(* Logix 5000 project; controller Carpenter_Meter_SCP vendor 1 type 14 code 217 rev 31.11; software revision 31.01; part 6 of 7 *)
(* tags used below, declared in another part *)
   AlwaysOff : BOOL;   // Always Off Bit
   CAR100_Flowpath : BOOL;   // Carpenter MLV CAR100 Flow Path (1=OK)
   CAR100_High_Pressure_SD : BOOL;   // Carpenter MLV CAR100 High Pressure Shutdown Status
   Carpenter_ISD_Command : BOOL;   // Carpenter/Hereford ISD Command from OCC (Through Pawnee)
   Carpenter_to_Pawnee_OK : BOOL;   // Carpenter to Pawnee Flow Path Permissive
   CC_Cust1_Flow_Permissive : BOOL;   // Customer #1 (MS8800) Flow Permissive to OCC
   CC_Cust1_Hi_WIOM : BOOL;   // Customer #1 High Water % Alarm to OCC
   CC_Cust1_Pump_Running : BOOL;   // Customer #1 (MS8800) Pump Running Status to OCC
   CC_Cust1_Ready : BOOL;   // Customer #1 (MS8800) Ready Status to OCC
   CC_Cust1_Shutin_Timer : REAL;   // Customer #1 Shutin Reset Time Left to OCC
   CC_Cust1_WIOM_Shutin : BOOL;   // Customer #1 Shutin Due to High High Water in Oil Monitor Alarm to OCC
   CC_Cust5_Flow_Permissive : BOOL;   // Customer #5 (MS8840) Flow Permissive to OCC
   CC_Cust5_Ready : BOOL;   // Customer #5 (MS8840) Ready Status to OCC
   CC_MS8800_Biocide_Flow : REAL;   // Meter Skid MS-8800 Biocide Flow Rate
   CC_MS8800_Biocide_Flow_SP : REAL;   // Meter Skid MS-8800 Biocide Flow Rate Setpoint
   CC_MS8800_CustPress : OCC_Analog;   // Meter Skid MS-8800 Customer Inlet Pressure to OCC
   CC_MS8810_CustPress : OCC_Analog;   // Meter Skid MS-8810 Customer Inlet Pressure to OCC
   CC_MS8820_CustPress : OCC_Analog;   // Meter Skid MS-8820 Customer Inlet Pressure to OCC
   CC_MS8830_CustPress : OCC_Analog;   // Meter Skid MS-8830 Customer Inlet Pressure to OCC
   CC_MS8840_Biocide_Flow : REAL;   // Meter Skid MS-8800 Biocide Flow Rate
   CC_MS8840_Biocide_Flow_SP : REAL;   // Meter Skid MS-8800 Biocide Flow Rate Setpoint
   CC_MS8840_CustPress : OCC_Analog;   // Meter Skid MS-8840 Customer Inlet Pressure to OCC
   CC_Pawnee_Flow_Path : BOOL;   // Flow Path to Pawnee
   CC_PV_0001 : OCC_CV;   // PV-0001
   CC_PV_0001_Flow_SP : DINT;   // Meter Skid MS8800 Inlet Control Valve Flow Setpoint
   CC_PV_0001_Press_SP : DINT;   // Meter Skid MS8800 Inlet Control Valve Press Setpoint
   CC_PV_0041 : OCC_CV;   // PV-0041
   CC_PV_0041_Flow_SP : DINT;   // Meter Skid MS8840 Inlet Control Valve Flow Setpoint
   CC_PV_0041_Press_SP : DINT;   // Meter Skid MS8800 Inlet Control Valve Press Setpoint
   CC_STA_Stop : BOOL;   // Station Stop Request Command from OCC
   CC_XI_0021 : BOOL;   // FGP Main PLC 24VDC Failure to OCC
   CC_XI_8800B : BOOL;   // MS8800 FGP 24VDC Failure to OCC
   CC_XI_8840B : BOOL;   // MS8840 FGP 24VDC Failure to OCC
   CC_YI_6000 : BOOL;   // UPS-6000 Utility Power Loss to OCC
   CC_YI_6001 : BOOL;   // UPS-6000 Fault
   cmd_reset_tmr : TIMER[8];   // General Use HMI Command Reset Timer
   Cust1_WIOM_Alarm : BOOL;   // Customer 1 WIOM Alarm
   Cust1_WIOM_Reset_Tmr : TIMER;   // Customer 1 Reset Timer for a WIOM Shutin
   Customer1_Flowpath_OK : BOOL;   // Customer #1 Flowpath Permissive (1 = OK)
   Customer1_Pump_Status : BOOL;   // Customer #1 Pump Running Status
   Customer1_Ready_Status : BOOL;   // Customer #1 Ready Status
   Customer5_Flowpath_OK : BOOL;   // Customer #5 Flowpath Permissive (1 = OK)
   Customer5_Ready_Status : BOOL;   // Customer #4 Ready Status
   fgp_deactivate_keysw : BOOL;   // Fire and Gas System Deactivated through Key Switch
   FGP_ESD : TGE_Alarm;   // ESD Shutdown from FGP (HS-0020A)
   FGP_Fire_Det : TGE_Alarm;   // Fire Shutdown from FGP (YSHH-0022)
   FGP_Gas_Det : TGE_Alarm;   // Hi Gas Shutdown from FGP (ASHH-0021)
   fgp_panel_reset : BOOL;   // FGP Panel Reset Pushbutton
   Hereford_Flowpath : BOOL;   // Pawnee Terminal Flow Path (1=OK)
   Hereford_High_Pressure_SD : BOOL;   // Hereford High Pressure Shutdown Status
   Hereford_OCC_HB_FAIL : BOOL;   // Pawnee High Pressure Shutdown Status
   HRF100_Flowpath : BOOL;   // Hereford MLV HRF100 Flow Path (1=OK)
   HRF100_High_Pressure_SD : BOOL;   // Hereford MLV HRF100 High Pressure Shutdown Status
   Main_FGP_24VDC_Fail : TGE_Alarm;   // Main PLC FGP 24VDC Fail (XS-0021)
   MS8800_Biocide_Flow_Fdbk_AOI : TGE_AI;   // Meter Skid MS-8800 Biocide Injection Rate Feedback
   MS8800_Biocide_Flow_SP : REAL;   // Meter Skid MS-8800 Biocide Flow Rate Gal/Day
   MS8800_Cust_Press : TGE_AI_UDT;   // Meter Skid MS-8800 Customer Inlet Pressure (Communicated from Cust)
   MS8800_FGP_24VDC_Fail : TGE_Alarm;   // Meter Skid MS-8800 FGP 24VDC Fail (XS-8800B)
   MS8800_Flow_Control : PID;   // Meter Skid MS8800 Flow Rate P&ID
   MS8800_Inlet_Press_Control : PID;   // Meter Skid MS8800 Customer Inlet Pressure P&ID
   MS8800_PCV_Pos_AOI : TGE_AI;   // Meter Skid MS-8800 Pressure Control Valve - Position Feedback (PCV-0001)
   MS8800_WIOM_Alarm : AnalogAlm;   // MS8800 Water In Oil Monitor Alarm (Setpoint Dictated by Tarrif)
   MS8840_Biocide_Flow_Fdbk_AOI : TGE_AI;   // Meter Skid MS-8840 Biocide Injection Rate Feedback
   MS8840_Biocide_Flow_SP : REAL;   // Meter Skid MS-8840 Biocide Flow Rate Gal/Day
   MS8840_Cust_Press : TGE_AI_UDT;   // Meter Skid MS-8840 Customer Inlet Pressure (Communicated from Cust)
   MS8840_FGP_24VDC_Fail : TGE_Alarm;   // Meter Skid MS-8840 FGP 24VDC Fail (XS-8840B)
   MS8840_Flow_Control : PID;   // Meter Skid MS8840 Flow Rate P&ID
   MS8840_Inlet_Press_Control : PID;   // Meter Skid MS8840 Customer Inlet Pressure P&ID
   MS8840_PCV_Pos_AOI : TGE_AI;   // Meter Skid MS-8840 Pressure Control Valve - Position Feedback (PCV-0041)
   ons_gen_use : BOOL[64];
   ovrd_disch_press : Override;   // Discharge Pressure Override
   ovrd_esd : Override;   // ESD Override
   ovrd_fire : Override;   // Fire Override
   ovrd_gas : Override;   // Gas Override
   Pawnee_ESD : BOOL;   // Pawnee Terminal ESD Signal (1=OK, 0 = ESD Active)
   Pawnee_Flowpath : BOOL;   // Pawnee Terminal Flow Path (1=OK)
   Pawnee_High_Pressure_SD : BOOL;   // Pawnee High Pressure Shutdown Status
   Pawnee_OCC_HB_FAIL : BOOL;   // Pawnee OCC HB Fail
   PV0001_Malf : TGE_Alarm;   // PV0001 Malfunction Alarm
   PV0001_Pos_Cmd : REAL;   // PCV-0001 Position Command
   PV0041_Malf : TGE_Alarm;   // PV0041 Malfunction Alarm
   PV0041_Pos_Cmd : REAL;   // PCV-0041 Position Command
   SCADA_HB_Fail_Alm : TGE_Alarm;   // SCADA Hearbeat Failure Alarm
   Sta_Stat : StaStatus;
   sta_stop : StaStartStop;   // Station Stop
   sta_stop_vlv_req : BOOL;   // Station Stop Valve Close Request
   Station_Disch_Press : TGE_AI_UDT;   // Station Discharge Pressure - Launcher Skid (PIT-1101)
   Test : BOOL;
   TU3000_HiHi_Lvl : TGE_Alarm;   // Sump Tank (TU-3000) Hi Hi Level Switch (LSHH-3000)
   TU3100_HiHi_Lvl : TGE_Alarm;   // Sump Tank (TU-3100) Hi Hi Level Switch (LSHH-3100)
   UPS_Fault : TGE_Alarm;   // UPS-6000 Fault (YS-6001)
   UPS_Online : TGE_Alarm;   // UPS-6000 Loss of AC Feed (YS-6000)
   valve_failure : BOOL;   // Valve Failure Override
   XV_0001 : BaseVLVLiquid;   // XV-0001
   XV_0041 : BaseVLVLiquid;   // XV-0041
   XV_1100 : BaseVLVLiquid;   // XV-1100
   XV_1101 : BaseVLVLiquid;   // XV-1101
(* OCC_Comms, continued *)

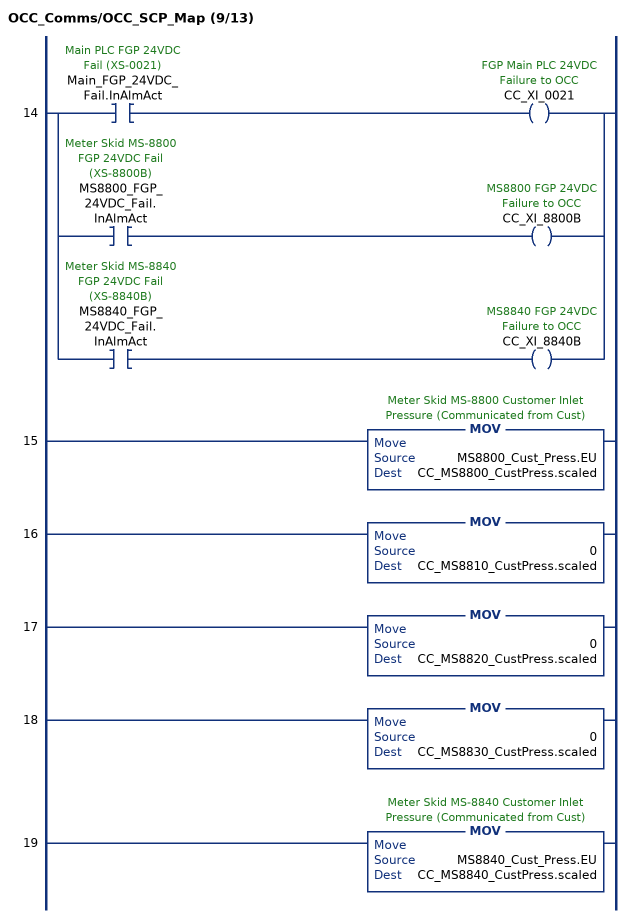
   [picture p98: OCC_Comms/OCC_SCP_Map rungs 14-19]
   14: [XIC(Main_FGP_24VDC_Fail.InAlmAct) OTE(CC_XI_0021) ,XIC(MS8800_FGP_24VDC_Fail.InAlmAct) OTE(CC_XI_8800B) ,XIC(MS8840_FGP_24VDC_Fail.InAlmAct) OTE(CC_XI_8840B) ];
   15: MOV(MS8800_Cust_Press.EU,CC_MS8800_CustPress.scaled);
   16: MOV(0,CC_MS8810_CustPress.scaled);
   17: MOV(0,CC_MS8820_CustPress.scaled);
   18: MOV(0,CC_MS8830_CustPress.scaled);
   19: MOV(MS8840_Cust_Press.EU,CC_MS8840_CustPress.scaled);
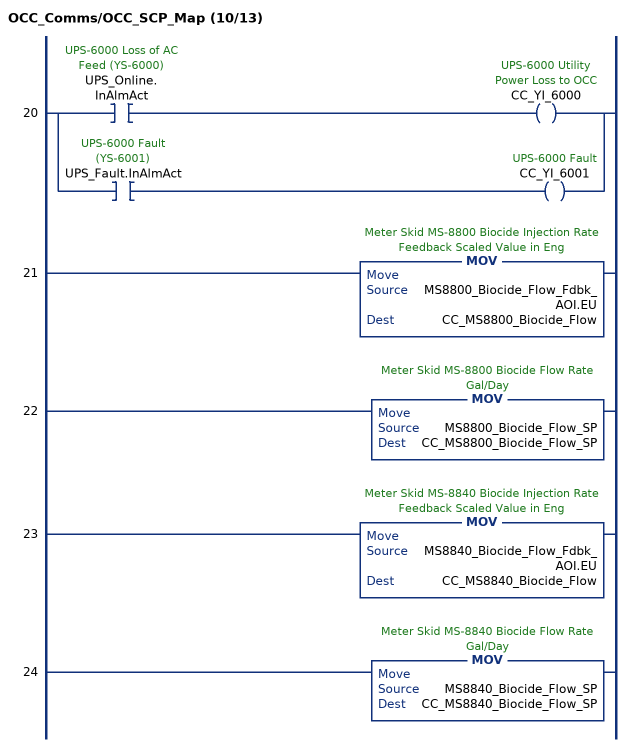
   20: [XIC(UPS_Online.InAlmAct) OTE(CC_YI_6000) ,XIC(UPS_Fault.InAlmAct) OTE(CC_YI_6001) ];
   21: MOV(MS8800_Biocide_Flow_Fdbk_AOI.EU,CC_MS8800_Biocide_Flow);
   22: MOV(MS8800_Biocide_Flow_SP,CC_MS8800_Biocide_Flow_SP);
   23: MOV(MS8840_Biocide_Flow_Fdbk_AOI.EU,CC_MS8840_Biocide_Flow);
   24: MOV(MS8840_Biocide_Flow_SP,CC_MS8840_Biocide_Flow_SP);
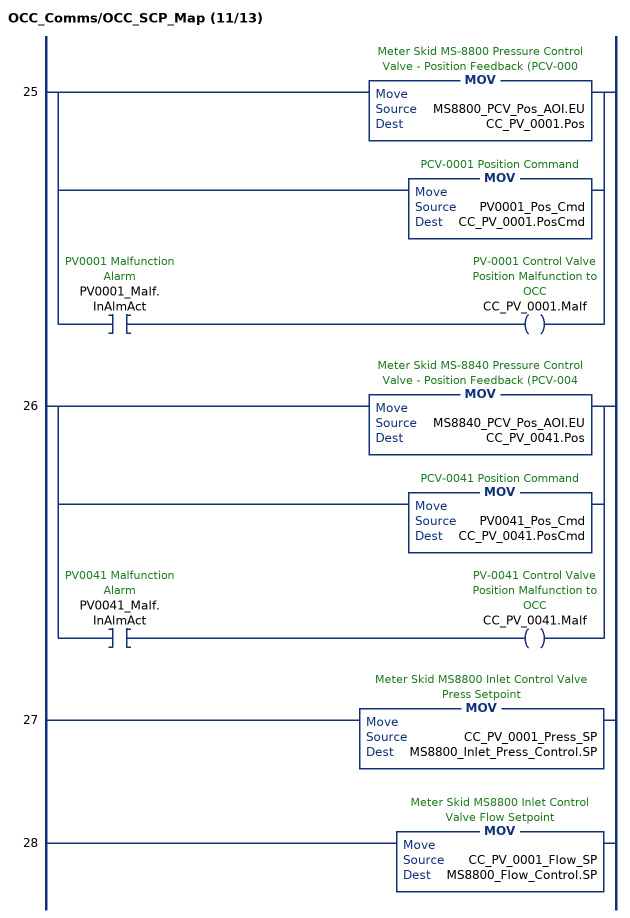
   25: [MOV(MS8800_PCV_Pos_AOI.EU,CC_PV_0001.Pos) ,MOV(PV0001_Pos_Cmd,CC_PV_0001.PosCmd) ,XIC(PV0001_Malf.InAlmAct) OTE(CC_PV_0001.Malf) ];
   26: [MOV(MS8840_PCV_Pos_AOI.EU,CC_PV_0041.Pos) ,MOV(PV0041_Pos_Cmd,CC_PV_0041.PosCmd) ,XIC(PV0041_Malf.InAlmAct) OTE(CC_PV_0041.Malf) ];
   27: MOV(CC_PV_0001_Press_SP,MS8800_Inlet_Press_Control.SP);
   28: MOV(CC_PV_0001_Flow_SP,MS8800_Flow_Control.SP);
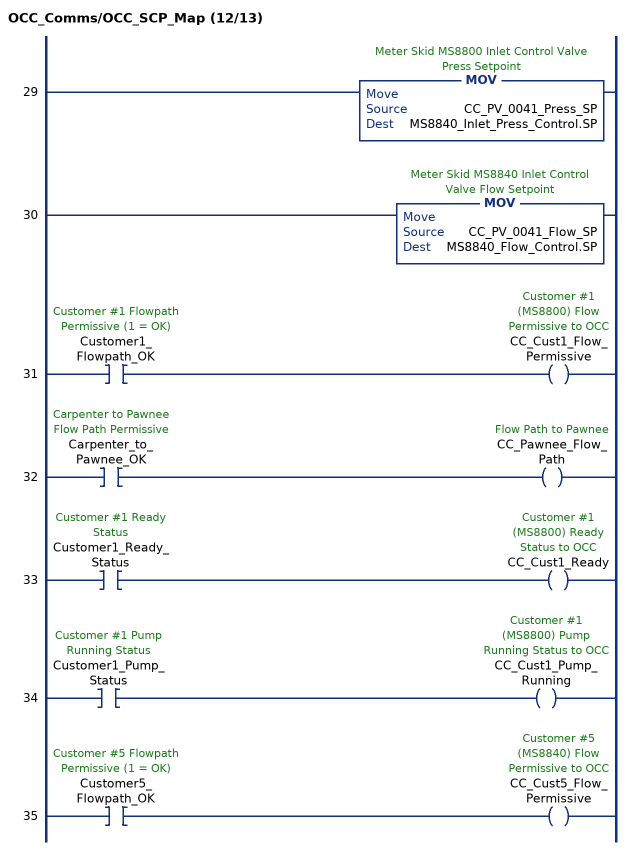
   29: MOV(CC_PV_0041_Press_SP,MS8840_Inlet_Press_Control.SP);
   30: MOV(CC_PV_0041_Flow_SP,MS8840_Flow_Control.SP);
   31: XIC(Customer1_Flowpath_OK)OTE(CC_Cust1_Flow_Permissive);
   32: XIC(Carpenter_to_Pawnee_OK)OTE(CC_Pawnee_Flow_Path);
   33: XIC(Customer1_Ready_Status)OTE(CC_Cust1_Ready);
   34: XIC(Customer1_Pump_Status)OTE(CC_Cust1_Pump_Running);
   35: XIC(Customer5_Flowpath_OK)OTE(CC_Cust5_Flow_Permissive);
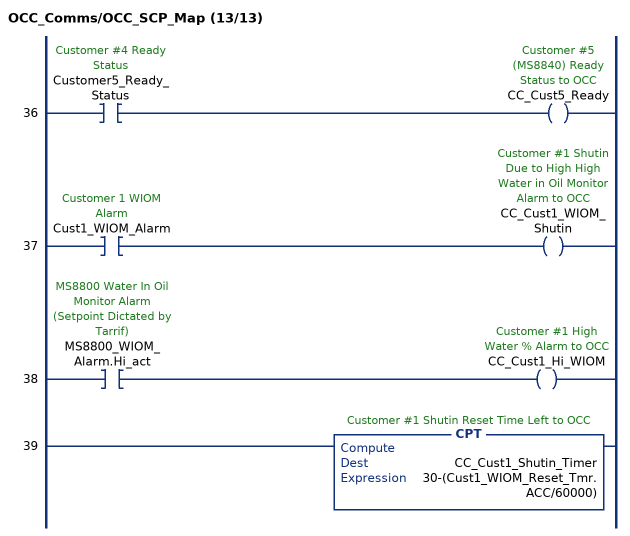
   36: XIC(Customer5_Ready_Status)OTE(CC_Cust5_Ready);
   37: XIC(Cust1_WIOM_Alarm)OTE(CC_Cust1_WIOM_Shutin);
   38: XIC(MS8800_WIOM_Alarm.Hi_act)OTE(CC_Cust1_Hi_WIOM);
   39: CPT(CC_Cust1_Shutin_Timer,30-(Cust1_WIOM_Reset_Tmr.ACC/60000));
END_ROUTINE
END_PROGRAM

PROGRAM Station_Control   (* main routine Station_Main *)

ROUTINE Flowpath   (* ladder *)
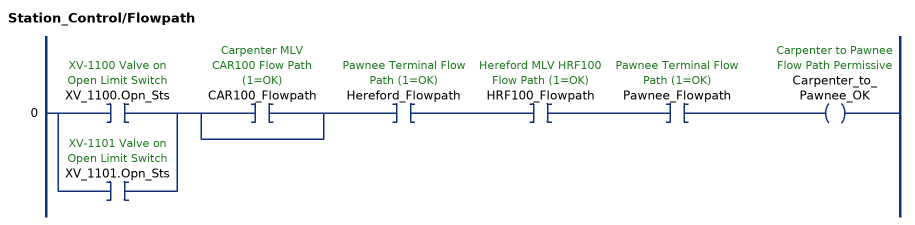
   0: [XIC(XV_1100.Opn_Sts) ,XIC(XV_1101.Opn_Sts) ][XIC(CAR100_Flowpath) ,]XIC(Hereford_Flowpath)XIC(HRF100_Flowpath)XIC(Pawnee_Flowpath)OTE(Carpenter_to_Pawnee_OK);
END_ROUTINE

ROUTINE Station_Main   (* ladder *)
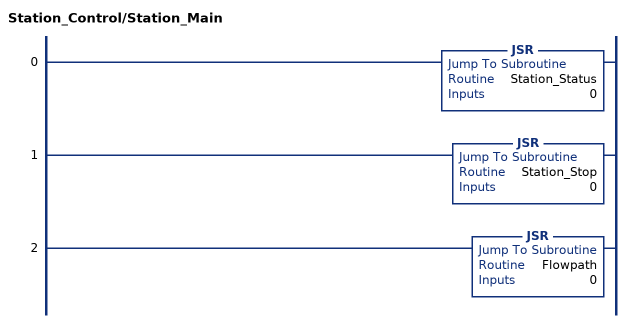
   0: JSR(Station_Status,0);
   1: JSR(Station_Stop,0);
   2: JSR(Flowpath,0);
END_ROUTINE

ROUTINE Station_Status   (* ladder *)
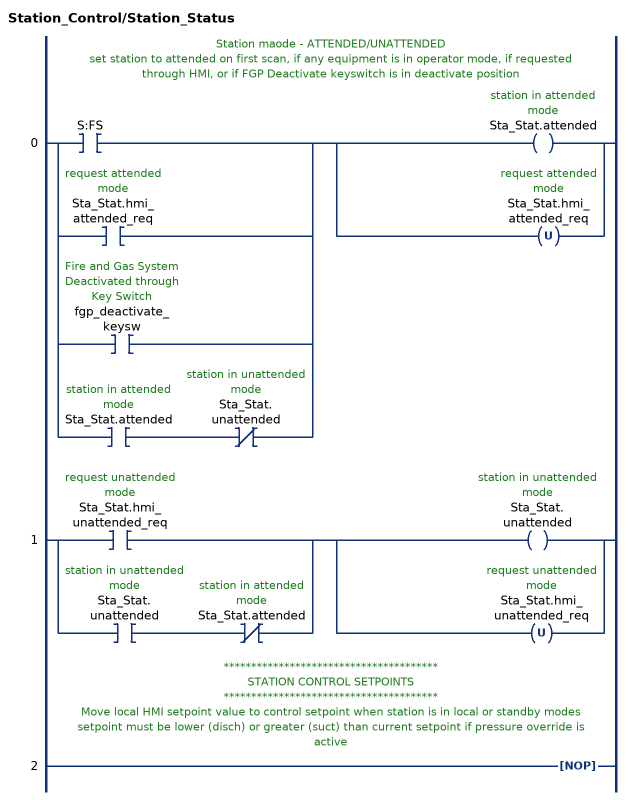
   // Station maode - ATTENDED/UNATTENDED
   // set station to attended on first scan, if any equipment is in operator mode, if requested through HMI, or if FGP Deactivate keyswitch is in deactivate position
   0: [XIC(S:FS) ,XIC(Sta_Stat.hmi_attended_req) ,XIC(fgp_deactivate_keysw) ,XIC(Sta_Stat.attended) XIO(Sta_Stat.unattended) ][OTE(Sta_Stat.attended) ,OTU(Sta_Stat.hmi_attended_req) ];
   1: [XIC(Sta_Stat.hmi_unattended_req) ,XIC(Sta_Stat.unattended) XIO(Sta_Stat.attended) ][OTE(Sta_Stat.unattended) ,OTU(Sta_Stat.hmi_unattended_req) ];
   // ***************************************
   // STATION CONTROL SETPOINTS
   // ***************************************
   // Move local HMI setpoint value to control setpoint when station is in local or standby modes
   // setpoint must be lower (disch) or greater (suct) than current setpoint if pressure override is active
   2: NOP();
END_ROUTINE

ROUTINE Station_Stop   (* ladder *)
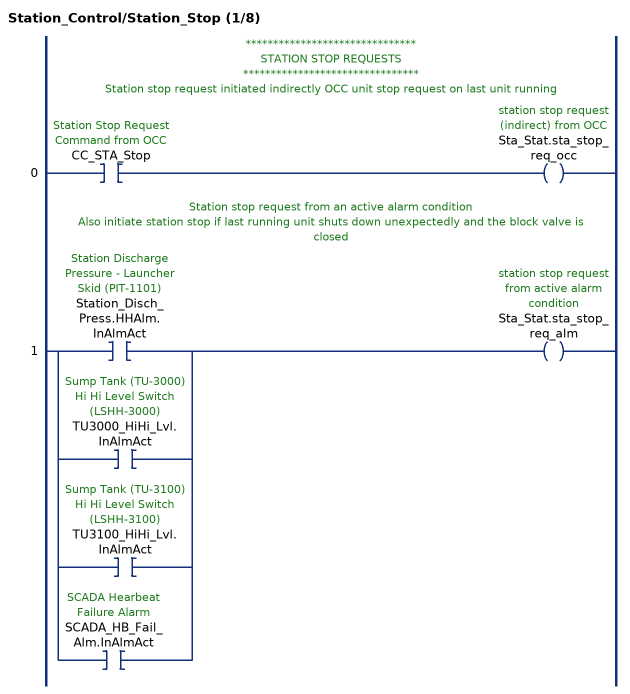
   // *******************************
   // STATION STOP REQUESTS
   // ********************************
   // Station stop request initiated indirectly OCC unit stop request on last unit running
   0: XIC(CC_STA_Stop)OTE(Sta_Stat.sta_stop_req_occ);
   // Station stop request from an active alarm condition
   // Also initiate station stop if last running unit shuts down unexpectedly and the block valve is closed
   1: [XIC(Station_Disch_Press.HHAlm.InAlmAct) ,XIC(TU3000_HiHi_Lvl.InAlmAct) ,XIC(TU3100_HiHi_Lvl.InAlmAct) ,XIC(SCADA_HB_Fail_Alm.InAlmAct) ]OTE(Sta_Stat.sta_stop_req_alm);
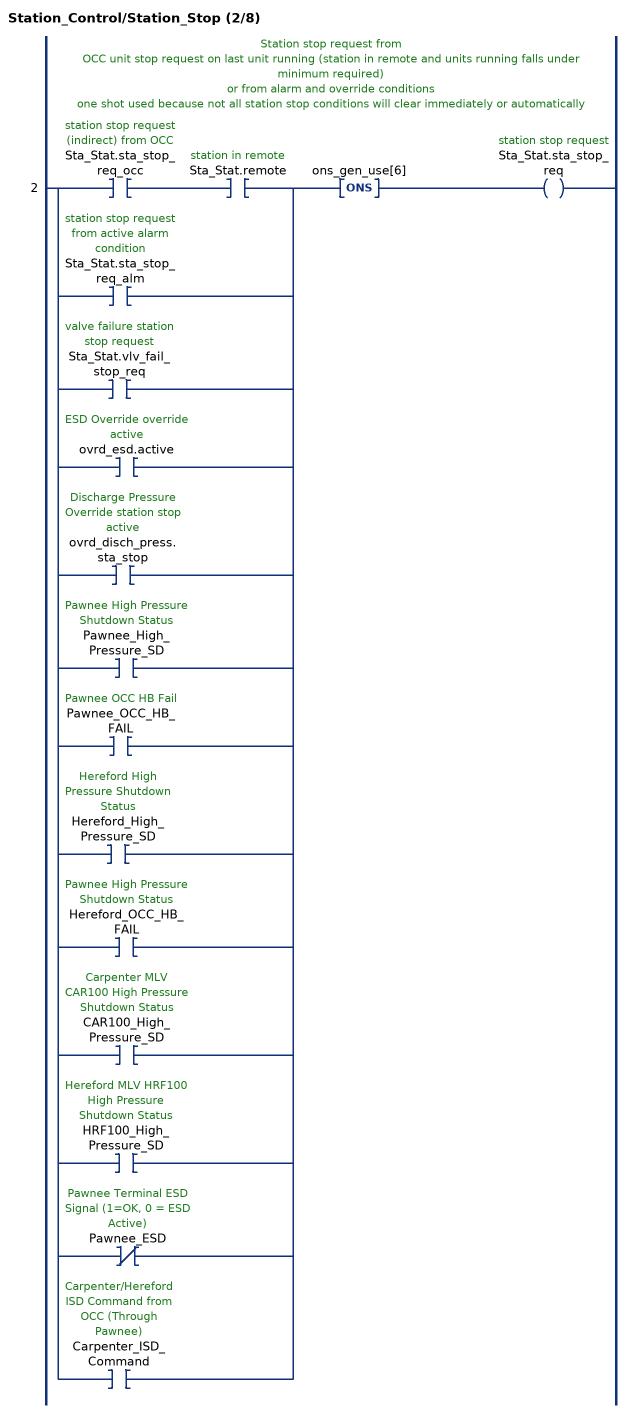
   // Station stop request from
   //  OCC unit stop request on last unit running (station in remote and units running falls under minimum required)
   // or from alarm and override conditions
   // one shot used because not all station stop conditions will clear immediately or automatically
   2: [XIC(Sta_Stat.sta_stop_req_occ) XIC(Sta_Stat.remote) ,XIC(Sta_Stat.sta_stop_req_alm) ,XIC(Sta_Stat.vlv_fail_stop_req) ,XIC(ovrd_esd.active) ,XIC(ovrd_disch_press.sta_stop) ,XIC(Pawnee_High_Pressure_SD) ,XIC(Pawnee_OCC_HB_FAIL) ,XIC(Hereford_High_Pressure_SD) ,XIC(Hereford_OCC_HB_FAIL) ,XIC(CAR100_High_Pressure_SD) ,XIC(HRF100_High_Pressure_SD) ,XIO(Pawnee_ESD) ,XIC(Carpenter_ISD_Command) ]ONS(ons_gen_use[6])OTE(Sta_Stat.sta_stop_req);
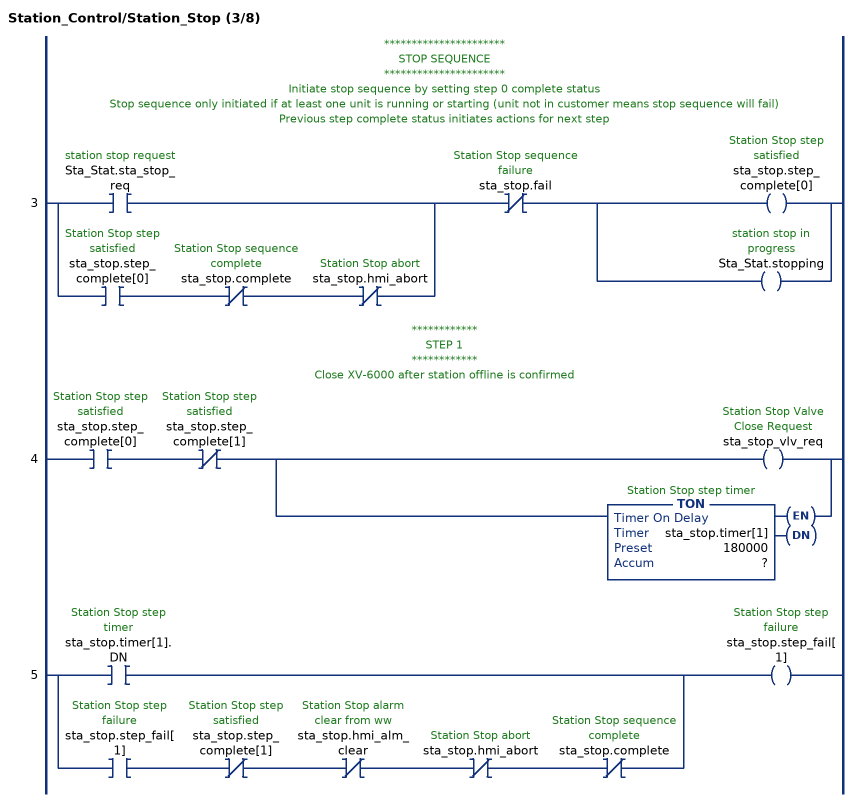
   // **********************
   // STOP SEQUENCE
   // **********************
   // Initiate stop sequence by setting step 0 complete status
   // Stop sequence only initiated if at least one unit is running or starting (unit not in customer means stop sequence will fail)
   // Previous step complete status initiates actions for next step
   3: [XIC(Sta_Stat.sta_stop_req) ,XIC(sta_stop.step_complete[0]) XIO(sta_stop.complete) XIO(sta_stop.hmi_abort) ]XIO(sta_stop.fail)[OTE(sta_stop.step_complete[0]) ,OTE(Sta_Stat.stopping) ];
   // ************
   // STEP 1
   // ************
   // Close XV-6000 after station offline is confirmed
   4: XIC(sta_stop.step_complete[0])XIO(sta_stop.step_complete[1])[OTE(sta_stop_vlv_req) ,TON(sta_stop.timer[1],?,?) ];
   5: [XIC(sta_stop.timer[1].DN) ,XIC(sta_stop.step_fail[1]) XIO(sta_stop.step_complete[1]) XIO(sta_stop.hmi_alm_clear) XIO(sta_stop.hmi_abort) XIO(sta_stop.complete) ]OTE(sta_stop.step_fail[1]);
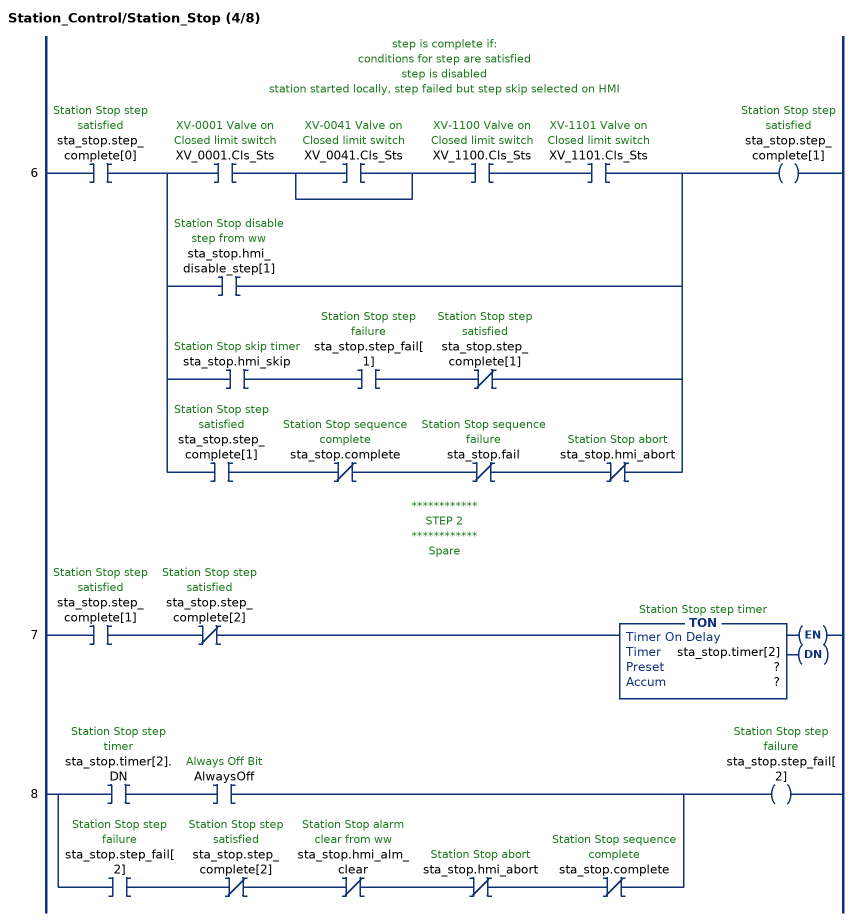
   // step is complete if:
   // conditions for step are satisfied
   // step is disabled
   // station started locally, step failed but step skip selected on HMI
   6: XIC(sta_stop.step_complete[0])[XIC(XV_0001.Cls_Sts) [XIC(XV_0041.Cls_Sts) ,] XIC(XV_1100.Cls_Sts) XIC(XV_1101.Cls_Sts) ,XIC(sta_stop.hmi_disable_step[1]) ,XIC(sta_stop.hmi_skip) XIC(sta_stop.step_fail[1]) XIO(sta_stop.step_complete[1]) ,XIC(sta_stop.step_complete[1]) XIO(sta_stop.complete) XIO(sta_stop.fail) XIO(sta_stop.hmi_abort) ]OTE(sta_stop.step_complete[1]);
   // ************
   // STEP 2
   // ************
   // Spare
   7: XIC(sta_stop.step_complete[1])XIO(sta_stop.step_complete[2])TON(sta_stop.timer[2],?,?);
   8: [XIC(sta_stop.timer[2].DN) XIC(AlwaysOff) ,XIC(sta_stop.step_fail[2]) XIO(sta_stop.step_complete[2]) XIO(sta_stop.hmi_alm_clear) XIO(sta_stop.hmi_abort) XIO(sta_stop.complete) ]OTE(sta_stop.step_fail[2]);
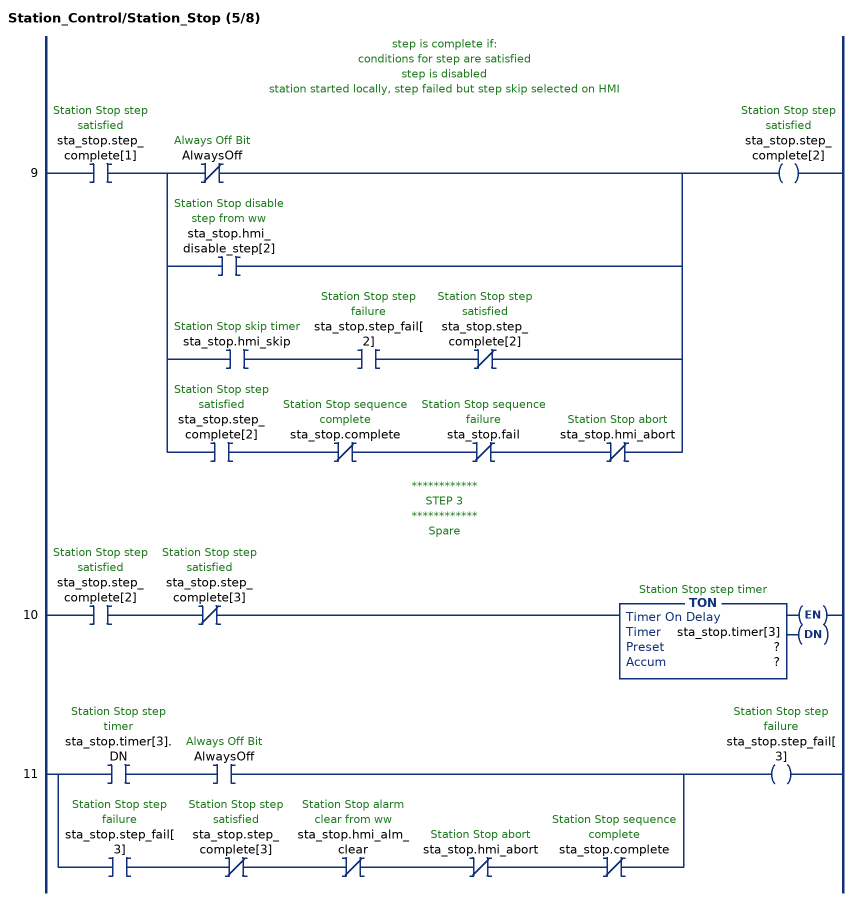
   // step is complete if:
   // conditions for step are satisfied
   // step is disabled
   // station started locally, step failed but step skip selected on HMI
   9: XIC(sta_stop.step_complete[1])[XIO(AlwaysOff) ,XIC(sta_stop.hmi_disable_step[2]) ,XIC(sta_stop.hmi_skip) XIC(sta_stop.step_fail[2]) XIO(sta_stop.step_complete[2]) ,XIC(sta_stop.step_complete[2]) XIO(sta_stop.complete) XIO(sta_stop.fail) XIO(sta_stop.hmi_abort) ]OTE(sta_stop.step_complete[2]);
   // ************
   // STEP 3
   // ************
   // Spare
   10: XIC(sta_stop.step_complete[2])XIO(sta_stop.step_complete[3])TON(sta_stop.timer[3],?,?);
   11: [XIC(sta_stop.timer[3].DN) XIC(AlwaysOff) ,XIC(sta_stop.step_fail[3]) XIO(sta_stop.step_complete[3]) XIO(sta_stop.hmi_alm_clear) XIO(sta_stop.hmi_abort) XIO(sta_stop.complete) ]OTE(sta_stop.step_fail[3]);
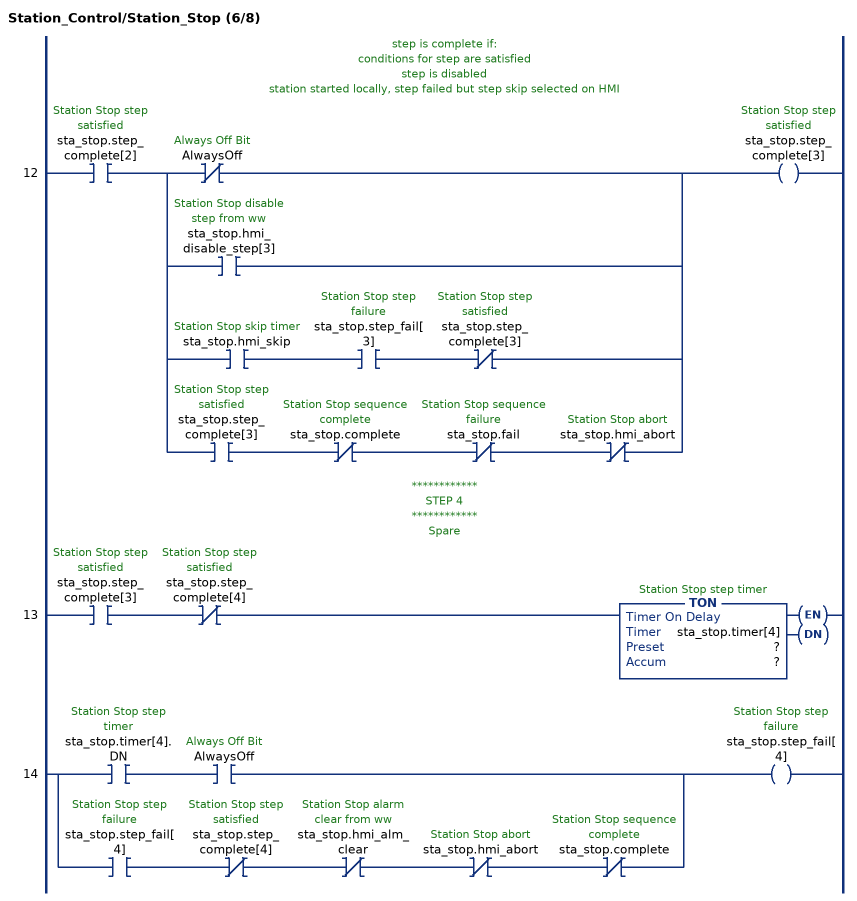
   // step is complete if:
   // conditions for step are satisfied
   // step is disabled
   // station started locally, step failed but step skip selected on HMI
   12: XIC(sta_stop.step_complete[2])[XIO(AlwaysOff) ,XIC(sta_stop.hmi_disable_step[3]) ,XIC(sta_stop.hmi_skip) XIC(sta_stop.step_fail[3]) XIO(sta_stop.step_complete[3]) ,XIC(sta_stop.step_complete[3]) XIO(sta_stop.complete) XIO(sta_stop.fail) XIO(sta_stop.hmi_abort) ]OTE(sta_stop.step_complete[3]);
   // ************
   // STEP 4
   // ************
   // Spare
   13: XIC(sta_stop.step_complete[3])XIO(sta_stop.step_complete[4])TON(sta_stop.timer[4],?,?);
   14: [XIC(sta_stop.timer[4].DN) XIC(AlwaysOff) ,XIC(sta_stop.step_fail[4]) XIO(sta_stop.step_complete[4]) XIO(sta_stop.hmi_alm_clear) XIO(sta_stop.hmi_abort) XIO(sta_stop.complete) ]OTE(sta_stop.step_fail[4]);
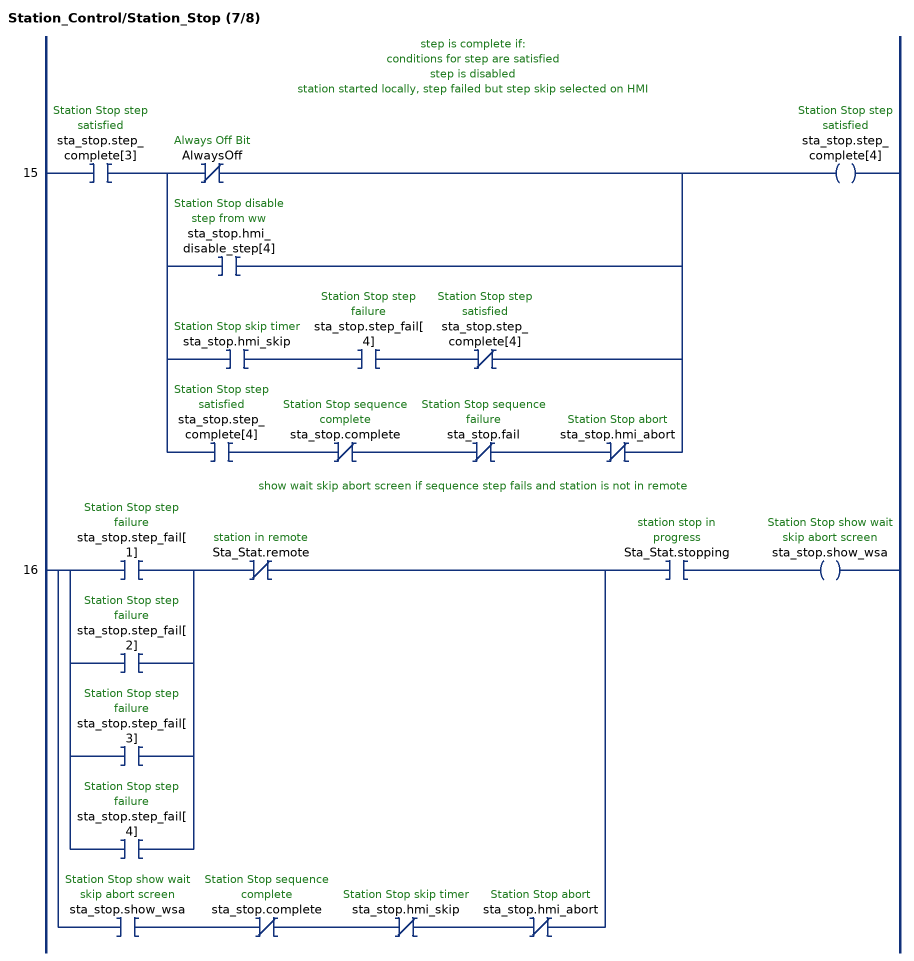
   // step is complete if:
   // conditions for step are satisfied
   // step is disabled
   // station started locally, step failed but step skip selected on HMI
   15: XIC(sta_stop.step_complete[3])[XIO(AlwaysOff) ,XIC(sta_stop.hmi_disable_step[4]) ,XIC(sta_stop.hmi_skip) XIC(sta_stop.step_fail[4]) XIO(sta_stop.step_complete[4]) ,XIC(sta_stop.step_complete[4]) XIO(sta_stop.complete) XIO(sta_stop.fail) XIO(sta_stop.hmi_abort) ]OTE(sta_stop.step_complete[4]);
   // show wait skip abort screen if sequence step fails and station is not in remote
   16: [[XIC(sta_stop.step_fail[1]) ,XIC(sta_stop.step_fail[2]) ,XIC(sta_stop.step_fail[3]) ,XIC(sta_stop.step_fail[4]) ] XIO(Sta_Stat.remote) ,XIC(sta_stop.show_wsa) XIO(sta_stop.complete) XIO(sta_stop.hmi_skip) XIO(sta_stop.hmi_abort) ]XIC(Sta_Stat.stopping)OTE(sta_stop.show_wsa);
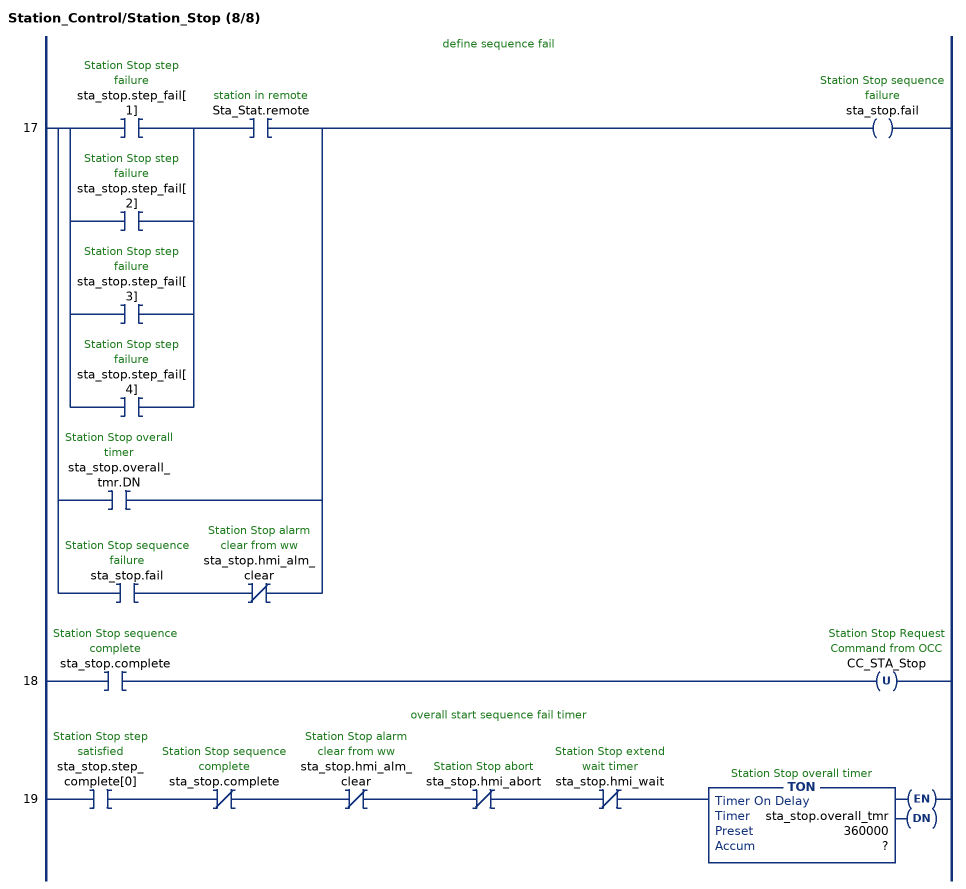
   // define sequence fail
   17: [[XIC(sta_stop.step_fail[1]) ,XIC(sta_stop.step_fail[2]) ,XIC(sta_stop.step_fail[3]) ,XIC(sta_stop.step_fail[4]) ] XIC(Sta_Stat.remote) ,XIC(sta_stop.overall_tmr.DN) ,XIC(sta_stop.fail) XIO(sta_stop.hmi_alm_clear) ]OTE(sta_stop.fail);
   18: XIC(sta_stop.complete)OTU(CC_STA_Stop);
   // overall start sequence fail timer
   19: XIC(sta_stop.step_complete[0])XIO(sta_stop.complete)XIO(sta_stop.hmi_alm_clear)XIO(sta_stop.hmi_abort)XIO(sta_stop.hmi_wait)TON(sta_stop.overall_tmr,?,?);
END_ROUTINE
END_PROGRAM

PROGRAM Station_Overrides   (* main routine Override_Main *)

ROUTINE Override_Main   (* ladder *)
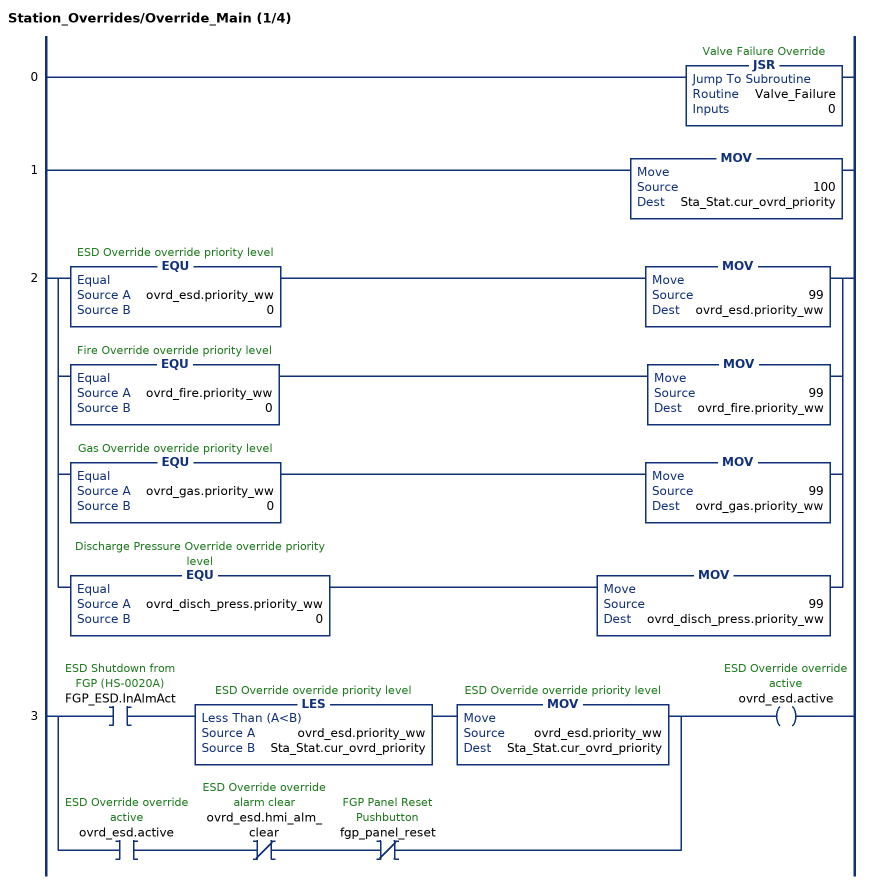
   0: JSR(Valve_Failure,0);
   1: MOV(100,Sta_Stat.cur_ovrd_priority);
   2: [EQU(ovrd_esd.priority_ww,0) MOV(99,ovrd_esd.priority_ww) ,EQU(ovrd_fire.priority_ww,0) MOV(99,ovrd_fire.priority_ww) ,EQU(ovrd_gas.priority_ww,0) MOV(99,ovrd_gas.priority_ww) ,EQU(ovrd_disch_press.priority_ww,0) MOV(99,ovrd_disch_press.priority_ww) ];
   3: [XIC(FGP_ESD.InAlmAct) LES(ovrd_esd.priority_ww,Sta_Stat.cur_ovrd_priority) MOV(ovrd_esd.priority_ww,Sta_Stat.cur_ovrd_priority) ,XIC(ovrd_esd.active) XIO(ovrd_esd.hmi_alm_clear) XIO(fgp_panel_reset) ]OTE(ovrd_esd.active);
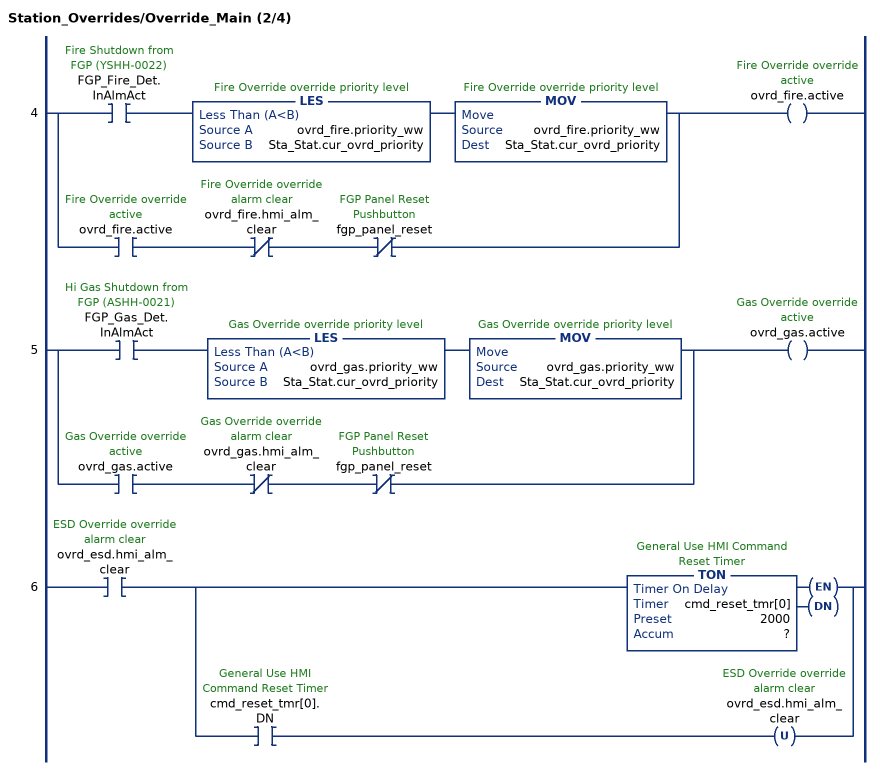
   4: [XIC(FGP_Fire_Det.InAlmAct) LES(ovrd_fire.priority_ww,Sta_Stat.cur_ovrd_priority) MOV(ovrd_fire.priority_ww,Sta_Stat.cur_ovrd_priority) ,XIC(ovrd_fire.active) XIO(ovrd_fire.hmi_alm_clear) XIO(fgp_panel_reset) ]OTE(ovrd_fire.active);
   5: [XIC(FGP_Gas_Det.InAlmAct) LES(ovrd_gas.priority_ww,Sta_Stat.cur_ovrd_priority) MOV(ovrd_gas.priority_ww,Sta_Stat.cur_ovrd_priority) ,XIC(ovrd_gas.active) XIO(ovrd_gas.hmi_alm_clear) XIO(fgp_panel_reset) ]OTE(ovrd_gas.active);
   6: XIC(ovrd_esd.hmi_alm_clear)[TON(cmd_reset_tmr[0],?,?) ,XIC(cmd_reset_tmr[0].DN) OTU(ovrd_esd.hmi_alm_clear) ];
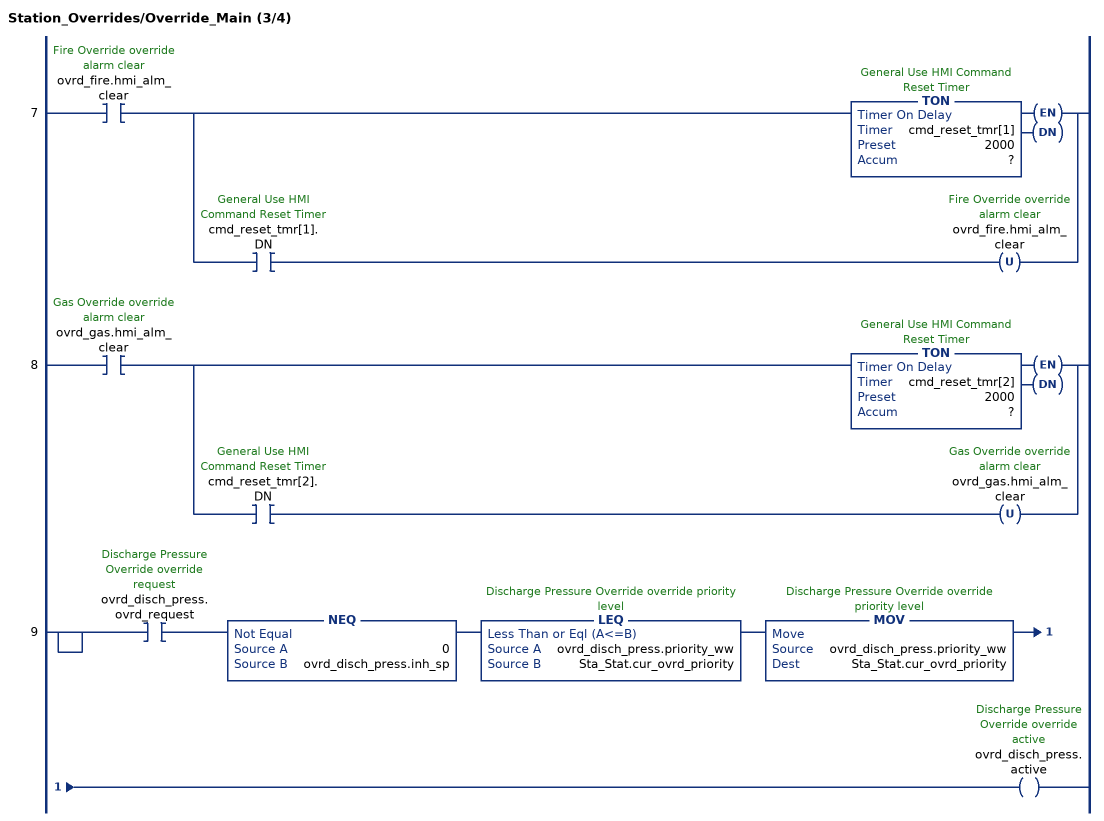
   7: XIC(ovrd_fire.hmi_alm_clear)[TON(cmd_reset_tmr[1],?,?) ,XIC(cmd_reset_tmr[1].DN) OTU(ovrd_fire.hmi_alm_clear) ];
   8: XIC(ovrd_gas.hmi_alm_clear)[TON(cmd_reset_tmr[2],?,?) ,XIC(cmd_reset_tmr[2].DN) OTU(ovrd_gas.hmi_alm_clear) ];
   9: [,]XIC(ovrd_disch_press.ovrd_request)NEQ(0,ovrd_disch_press.inh_sp)LEQ(ovrd_disch_press.priority_ww,Sta_Stat.cur_ovrd_priority)MOV(ovrd_disch_press.priority_ww,Sta_Stat.cur_ovrd_priority)OTE(ovrd_disch_press.active);
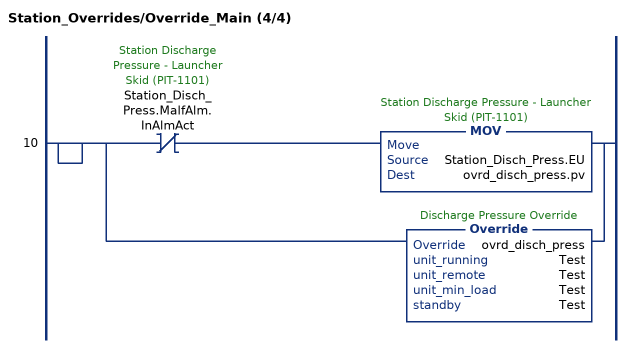
   10: [,][XIO(Station_Disch_Press.MalfAlm.InAlmAct) MOV(Station_Disch_Press.EU,ovrd_disch_press.pv) ,Override(ovrd_disch_press,Test,Test,Test,Test) ];
END_ROUTINE
